FUNCTION IsNotNull : BOOL
VAR_INPUT
	anyPtrType		: ANY;
END_VAR

IF anyPtrType.diSize = SIZEOF(POINTER TO BYTE) THEN
	IsNotNull := anyPtrType.pValue^ <> 0;
END_IF

END_FUNCTION

(* stored: Version 1.1.0.1
   POU IsNotNull: Id {70442020-8eef-4670-a400-c8f68f316235}, SpecialFunc None *)
